FUNCTION_BLOCK FB_Co2ConsumptionHandler
VAR_INPUT
	meanFlow : REAL;
	flowControlParameters : ST_FlowControlParameters;
	resetInput : BOOL;
END_VAR
VAR_OUTPUT
	consumedCo2Amount : REAL;
END_VAR
VAR
	consumptionCalculator : FB_ConsumptionCalculator;
END_VAR


IF flowControlParameters.startConsumptionCalculationWithAvg THEN 
	consumptionCalculator.calculate(
								start := NOT resetInput,
								valuePerSec := meanFlow/60,
								intervalS := flowControlParameters.movingAvgShiftIntervalSecs,
								dtime := T#10MS);
END_IF
							
consumedCo2Amount := consumptionCalculator.sum;

IF resetInput THEN
	consumptionCalculator.reset();
END_IF

END_FUNCTION_BLOCK

(* stored: Version 1.1.0.1, ProductVersion 3.1.4024.9
   POU FB_Co2ConsumptionHandler: Id {21a94a87-e497-4368-ab09-e83da1788240}, SpecialFunc None *)
